// TwinCAT 3 PLC project PLC
// ProgramVersion: 3.1.4023.0
// libraries:
//   Tc2_MC2, * (Beckhoff Automation GmbH)
//   Tc2_Standard, * (Beckhoff Automation GmbH)
//   Tc2_System, * (Beckhoff Automation GmbH)
//   Tc2_Utilities, * (Beckhoff Automation GmbH)
//   Tc3_Module, * (Beckhoff Automation GmbH)
// project tree:
//   DUTs/ E_AxisId.TcDUT
//   GVLs/ GVL_Global.TcGVL, GVL_IO.TcGVL
//   / PlcTask.TcTTO
//   POUs/ MAIN.TcPOU
//   POUs/Motion/ FB_Servo.TcPOU, Motion.TcPOU
// real-time tasks:
//   TASK PlcTask: cycle T#10ms, priority 20, ADS port 350
// motion (NC):
//   TASK NC-Task 1 SAF: cycle T#2ms, priority 4, ADS port 501
//   TASK NC-Task 1 SVB: cycle T#10ms, priority 8, ADS port 511
//   AXIS Axis 1 (id 1)
//     OtherSettings: AllowMotionCmdToSlave=true
//     encoder EncType=1
//     drive DrvType=5
//       Analog: TorqueSetpointScale=10, ScaleFactorActTorque=0.1
//       TimeComp: TaskDelayCycles=1
//     controller CtrType=1
//       CtrPara: PriorControlFactor=1
//         Observer: BandWidth=20
//   AXIS Axis 2 (id 2)
//     OtherSettings: AllowMotionCmdToSlave=true
//     encoder EncType=1
//     drive DrvType=5
//       Analog: TorqueSetpointScale=10, ScaleFactorActTorque=0.1
//       TimeComp: TaskDelayCycles=1
//     controller CtrType=1
//       CtrPara: PriorControlFactor=1
//         Observer: BandWidth=20

CONFIGURATION PLC
    RESOURCE PLC ON TwinCAT3
        TASK PlcTask(INTERVAL := T#10ms, PRIORITY := 20);
        PROGRAM MAIN WITH PlcTask : MAIN;
    END_RESOURCE
END_CONFIGURATION

// ---- DUTs/E_AxisId.TcDUT
{attribute 'toString'}
TYPE E_AxisId :
(
	enum_member := 0,
	eAxis1		:= 1,
	eAxis2		:= 2
	
);
END_TYPE

// ---- GVLs/GVL_Global.TcGVL
VAR_GLOBAL

	
END_VAR

// ---- GVLs/GVL_IO.TcGVL
{attribute 'qualified_only'}
VAR_GLOBAL CONSTANT
	cNrOfAxes:					INT := 2;
	
END_VAR

VAR_GLOBAL
	stAxisRef:					ARRAY[1..cNrOfAxes] OF AXIS_REF;
	
END_VAR

// ---- POUs/MAIN.TcPOU
PROGRAM MAIN
VAR
END_VAR

END_PROGRAM

// ---- POUs/Motion/FB_Servo.TcPOU
FUNCTION_BLOCK FB_Servo

(*
	Beckhoff motion
*)

VAR_INPUT
	stAxis:			AXIS_REF;
	
	fOverride:		LREAL;
	
END_VAR

VAR_OUTPUT
END_VAR

VAR
// instance data
	fbPower:		MC_POWER;

END_VAR




// MC_POWER
fbPower(
	Axis:= stAxis, 
	Enable:= TRUE, 
	Enable_Positive:= TRUE, 
	Enable_Negative:= TRUE, 
	Override:= fOverride, 
	BufferMode:= , 
	Options:= , 
	Status=> , 
	Busy=> , 
	Active=> , 
	Error=> , 
	ErrorID=> );

END_FUNCTION_BLOCK

// ---- POUs/Motion/Motion.TcPOU
PROGRAM Motion
VAR
	
// motion
	fOverride:		LREAL := 100.0;

// instance data
	fbServo:		ARRAY[1..GVL_IO.cNrOfAxes] OF FB_Servo;
		
END_VAR


// axis 1
	fbServo[eAxis1](stAxis:= GVL_IO.stAxisRef[eAxis1],
		fOverride:= fOverride);

// axis 2
	fbServo[eAxis2](stAxis:= GVL_IO.stAxisRef[eAxis2],
		fOverride:= fOverride);

END_PROGRAM
